// TIA Portal V16 program export: 1 tag tables, 0 data types, 2 data blocks, 2 code blocks (in call order from the OBs), 5 instance data blocks

VAR_GLOBAL   // PLC tag table "Default tag table"
   System_Byte AT %MB100 : Byte;
   FirstScan AT %M100.0 : Bool;
   DiagStatusUpdate AT %M100.1 : Bool;
   AlwaysTRUE AT %M100.2 : Bool;
   AlwaysFALSE AT %M100.3 : Bool;
   "System_Byte(1)" AT %MB1 : Byte;
   Clock_Byte AT %MB101 : Byte;
   Clock_10Hz AT %M101.0 : Bool;
   Clock_5Hz AT %M101.1 : Bool;
   "Clock_2.5Hz" AT %M101.2 : Bool;
   Clock_2Hz AT %M101.3 : Bool;
   "Clock_1.25Hz" AT %M101.4 : Bool;
   Clock_1Hz AT %M101.5 : Bool;
   "Clock_0.625Hz" AT %M101.6 : Bool;
   "Clock_0.5Hz" AT %M101.7 : Bool;
END_VAR

DATA_BLOCK "Data"   // DB6
{ S7_Optimized_Access := 'TRUE' }
VERSION : 0.1
// stored: AutoNumber true, DBAccessibleFromOPCUA true, IsOnlyStoredInLoadMemory false, IsRetainMemResEnabled false, IsWriteProtectedInAS false, MemoryReserve 100
   VAR
      send : Array[0..3] of Int;
      recv : Array[0..1] of Int;
   END_VAR
BEGIN
   send[0] := 2;
   send[1] := 6;
   send[2] := 8;
   send[3] := 12;
   recv[0] := 5;
   recv[1] := 7;
END_DATA_BLOCK

DATA_BLOCK "connect"   // DB4
{ S7_Optimized_Access := 'TRUE' }
VERSION : 0.1
// stored: AutoNumber true, DBAccessibleFromOPCUA true, IsOnlyStoredInLoadMemory false, IsRetainMemResEnabled false, IsWriteProtectedInAS false, MemoryReserve 100
   VAR
      req : Bool;
      disconnect : Bool;
      send { S7_SetPoint := 'True'} : TCON_IP_v4;
      recv : TCON_IP_v4;
   END_VAR
BEGIN
   send.InterfaceId := 64;
   send.ID := 1;
   send.ConnectionType := 11;
   send.ActiveEstablished := true;
   send.RemoteAddress.ADDR[1] := 192;
   send.RemoteAddress.ADDR[2] := 168;
   send.RemoteAddress.ADDR[3] := 1;
   send.RemoteAddress.ADDR[4] := 11;
   send.RemotePort := 502;
   send.LocalPort := 502;
   recv.InterfaceId := 64;
   recv.ID := 2;
   recv.ConnectionType := 11;
   recv.ActiveEstablished := true;
   recv.RemoteAddress.ADDR[1] := 192;
   recv.RemoteAddress.ADDR[2] := 168;
   recv.RemoteAddress.ADDR[3] := 1;
   recv.RemoteAddress.ADDR[4] := 11;
   recv.RemotePort := 502;
   recv.LocalPort := 502;
END_DATA_BLOCK

ORGANIZATION_BLOCK "Main"   // OB1, LAD, ProgramCycle
TITLE = "Main Program Sweep (Cycle)"
{ S7_Optimized_Access := 'TRUE' }
VERSION : 0.1
// stored: AutoNumber true, IsIECCheckEnabled false, SetENOAutomatically false
   VAR_INPUT
      Initial_Call : Bool;   // Initial call of this OB
      Remanence : Bool;   // =True, if remanent data are available
   END_VAR
BEGIN

REGION Network 1
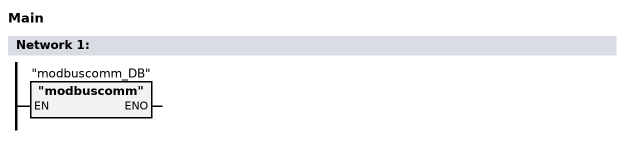
   RUNG wire#powerrail
      "modbuscomm_DB"()
   END_RUNG
   // the same network as SCL:
   "modbuscomm_DB"();   // "modbuscomm"
END_REGION
END_ORGANIZATION_BLOCK

FUNCTION_BLOCK "modbuscomm"   // FB1, LAD
{ S7_Optimized_Access := 'TRUE' }
VERSION : 0.1
// stored: AutoNumber true, IsIECCheckEnabled false, IsRetainMemResEnabled false, MemoryReserve 100, SetENOAutomatically false, UDAEnableTagReadback false
   VAR_TEMP
      tag1 : Bool;
      tag2 : Bool;
   END_VAR
BEGIN

REGION Network 1
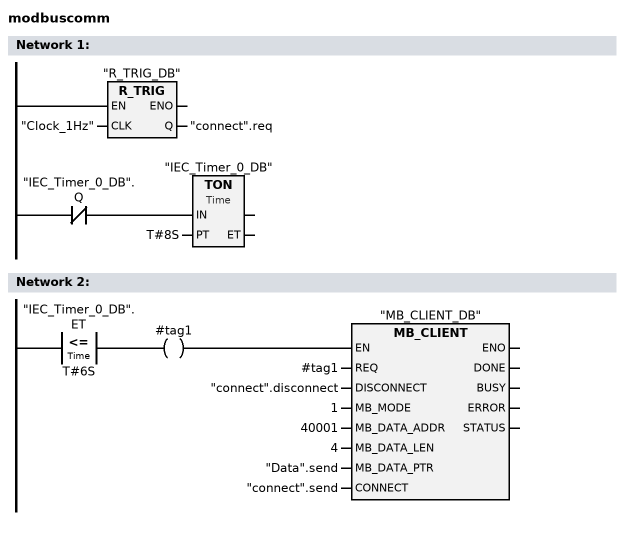
   RUNG wire#powerrail
      "R_TRIG_DB".R_TRIG(CLK := "Clock_1Hz", Q => "connect".req)
   END_RUNG
   RUNG wire#powerrail
      I_Contact( "IEC_Timer_0_DB".Q )
      { S7_Templates := "time_type := Time" } "IEC_Timer_0_DB".TON(pt := T#8S, et =>)
   END_RUNG
   // the same network as SCL:
   "R_TRIG_DB"(CLK := "Clock_1Hz", Q => "connect".req);   // R_TRIG
   "IEC_Timer_0_DB".TON(IN := NOT "IEC_Timer_0_DB".Q, PT := T#8S);
END_REGION

REGION Network 2
   RUNG wire#powerrail
      { S7_Templates := "SrcType := Time" } LE_Contact(in1 := "IEC_Timer_0_DB".ET, in2 := T#6S)
      Coil( #tag1 )
      "MB_CLIENT_DB".MB_CLIENT(REQ := #tag1, DISCONNECT := "connect".disconnect, MB_MODE := 1, MB_DATA_ADDR := 40001, MB_DATA_LEN := 4, MB_DATA_PTR := "Data".send, CONNECT := "connect".send, DONE =>, BUSY =>, ERROR =>, STATUS =>)
   END_RUNG
   // the same network as SCL:
   #tag1 := "IEC_Timer_0_DB".ET <= T#6S;
   IF #tag1 THEN
       "MB_CLIENT_DB"(REQ := #tag1,   // MB_CLIENT
                      DISCONNECT := "connect".disconnect,
                      MB_MODE := 1,
                      MB_DATA_ADDR := 40001,
                      MB_DATA_LEN := 4,
                      MB_DATA_PTR := "Data".send,
                      CONNECT := "connect".send);
   END_IF;
END_REGION
END_FUNCTION_BLOCK

DATA_BLOCK "modbuscomm_DB"   // DB7
VERSION : 0.1
// stored: AutoNumber true, DBAccessibleFromOPCUA true, InstanceOfName modbuscomm, InstanceOfType FB
"modbuscomm"
BEGIN
END_DATA_BLOCK

DATA_BLOCK "IEC_Timer_0_DB"   // DB5
{ S7_Optimized_Access := 'TRUE' }
// stored: AutoNumber true, DBAccessibleFromOPCUA true, InstanceOfName IEC_TIMER, OfSystemLibElement IEC_TIMER, OfSystemLibVersion 1.0
"IEC_TIMER"
   // VAR
   //    PT : Time;
   //    ET { ExternalWritable := 'False'} : Time;
   //    IN : Bool;
   //    Q { ExternalWritable := 'False'} : Bool;
   // END_VAR
BEGIN
END_DATA_BLOCK

DATA_BLOCK "MB_CLIENT_DB"   // DB1
// stored: AutoNumber true, DBAccessibleFromOPCUA true, InstanceOfName MB_CLIENT, OfSystemLibElement MB_CLIENT, OfSystemLibVersion 5.2
"MB_CLIENT"
   // VAR_INPUT
   //    REQ : Bool;
   //    DISCONNECT : Bool;
   //    MB_MODE : USInt;
   //    MB_DATA_ADDR : UDInt;
   //    MB_DATA_LEN : UInt;
   // END_VAR
   // VAR_OUTPUT
   //    DONE : Bool;
   //    BUSY : Bool;
   //    ERROR : Bool;
   //    STATUS { ExternalVisible := 'False'} : Word;
   // END_VAR
   // VAR_IN_OUT
   //    MB_DATA_PTR : Variant;
   //    CONNECT : Variant;
   // END_VAR
   // VAR
   //    TCON { S7_SetPoint := 'True'} : TCON;
   //    TDISCON { S7_SetPoint := 'True'} : TDISCON;
   //    TSEND { S7_SetPoint := 'True'} : TSEND;
   //    TRECEIVE { S7_SetPoint := 'True'} : TRCV;
   //    TRESET { S7_SetPoint := 'True'} : T_RESET;
   //    TDIAG { S7_SetPoint := 'True'} : T_DIAG;
   //    TDIAG_Status { S7_SetPoint := 'True'} : TDiag_Status;
   //    Blocked_Proc_Timeout : Real;
   //    Rcv_Timeout : Real;
   //    MB_Unit_ID : Byte;
   //    MB_Transaction_ID : Word;
   //    MB_State { ExternalWritable := 'False'} : Word;
   //    SAVED_MB_DATA_ADDR : UDInt;
   //    SAVED_DATA_LEN : UInt;
   //    SAVED_MB_MODE : USInt;
   //    Connection_ID : Word;
   //    Retries : Word;
   //    TEMP_DATA { ExternalWritable := 'False'} : Array[1..263] of Byte;
   //    rcv_timer { ExternalAccessible := 'False'; ExternalVisible := 'False'; ExternalWritable := 'False'; S7_SetPoint := 'True'} : TON_TIME;
   //    wd_timer { ExternalAccessible := 'False'; ExternalVisible := 'False'; ExternalWritable := 'False'; S7_SetPoint := 'True'} : TON_TIME;
   //    Connected : Bool;
   //    Active { ExternalWritable := 'False'} : Bool;
   //    BytesReceived : UDInt;
   // END_VAR
BEGIN
END_DATA_BLOCK

DATA_BLOCK "MB_CLIENT_DB_1"   // DB2
// stored: AutoNumber true, DBAccessibleFromOPCUA true, InstanceOfName MB_CLIENT, OfSystemLibElement MB_CLIENT, OfSystemLibVersion 5.2
"MB_CLIENT"
   // VAR_INPUT
   //    REQ : Bool;
   //    DISCONNECT : Bool;
   //    MB_MODE : USInt;
   //    MB_DATA_ADDR : UDInt;
   //    MB_DATA_LEN : UInt;
   // END_VAR
   // VAR_OUTPUT
   //    DONE : Bool;
   //    BUSY : Bool;
   //    ERROR : Bool;
   //    STATUS { ExternalVisible := 'False'} : Word;
   // END_VAR
   // VAR_IN_OUT
   //    MB_DATA_PTR : Variant;
   //    CONNECT : Variant;
   // END_VAR
   // VAR
   //    TCON { S7_SetPoint := 'True'} : TCON;
   //    TDISCON { S7_SetPoint := 'True'} : TDISCON;
   //    TSEND { S7_SetPoint := 'True'} : TSEND;
   //    TRECEIVE { S7_SetPoint := 'True'} : TRCV;
   //    TRESET { S7_SetPoint := 'True'} : T_RESET;
   //    TDIAG { S7_SetPoint := 'True'} : T_DIAG;
   //    TDIAG_Status { S7_SetPoint := 'True'} : TDiag_Status;
   //    Blocked_Proc_Timeout : Real;
   //    Rcv_Timeout : Real;
   //    MB_Unit_ID : Byte;
   //    MB_Transaction_ID : Word;
   //    MB_State { ExternalWritable := 'False'} : Word;
   //    SAVED_MB_DATA_ADDR : UDInt;
   //    SAVED_DATA_LEN : UInt;
   //    SAVED_MB_MODE : USInt;
   //    Connection_ID : Word;
   //    Retries : Word;
   //    TEMP_DATA { ExternalWritable := 'False'} : Array[1..263] of Byte;
   //    rcv_timer { ExternalAccessible := 'False'; ExternalVisible := 'False'; ExternalWritable := 'False'; S7_SetPoint := 'True'} : TON_TIME;
   //    wd_timer { ExternalAccessible := 'False'; ExternalVisible := 'False'; ExternalWritable := 'False'; S7_SetPoint := 'True'} : TON_TIME;
   //    Connected : Bool;
   //    Active { ExternalWritable := 'False'} : Bool;
   //    BytesReceived : UDInt;
   // END_VAR
BEGIN
END_DATA_BLOCK

DATA_BLOCK "R_TRIG_DB"   // DB3
// stored: AutoNumber true, DBAccessibleFromOPCUA true, InstanceOfName R_TRIG, OfSystemLibElement R_TRIG, OfSystemLibVersion 1.0
"R_TRIG"
   // VAR_INPUT
   //    CLK : Bool;
   // END_VAR
   // VAR_OUTPUT
   //    Q : Bool;
   // END_VAR
   // VAR
   //    Stat_Bit : Bool;
   // END_VAR
BEGIN
END_DATA_BLOCK
